{attribute 'TcGenerated'}
{attribute 'no-analysis'}
{attribute 'linkalways'}
// This function has been automatically generated from the project information.
VAR_GLOBAL CONSTANT
	{attribute 'const_non_replaced'}
	stLibVersion_HomePLC_Alarm_Manager : ST_LibVersion := (iMajor := 1, iMinor := 0, iBuild := 5, iRevision := 0, nFlags := 0, sVersion := '1.0.5');
END_VAR

(* stored: Version 1.1.0.1, ProductVersion 3.1.4024.12
   GVL Global_Version: Id {c2877152-2c8e-4121-9a8a-88ccc26e4604} *)
